(* Logix 5000 project; controller Week_4_PLC_1_Compare_Instructions Emulate 5570 rev 30.11; software revision 30.01 *)

TASK MainTask (continuous, watchdog 500 ms) : MainProgram

MODULES
   Local : Emulate 5570 (ICP 2, rev 30.11)
END_MODULES

PROGRAM MainProgram   (* main routine MainRoutine *)
VAR
   Counter : COUNTER := (PRE := 10);
   Output1 : BOOL;
   Output2 : BOOL;
   Output3 : BOOL;
   Output4 : BOOL;
   Output5 : BOOL;
   PB1 : BOOL;
END_VAR

ROUTINE MainRoutine   (* ladder *)
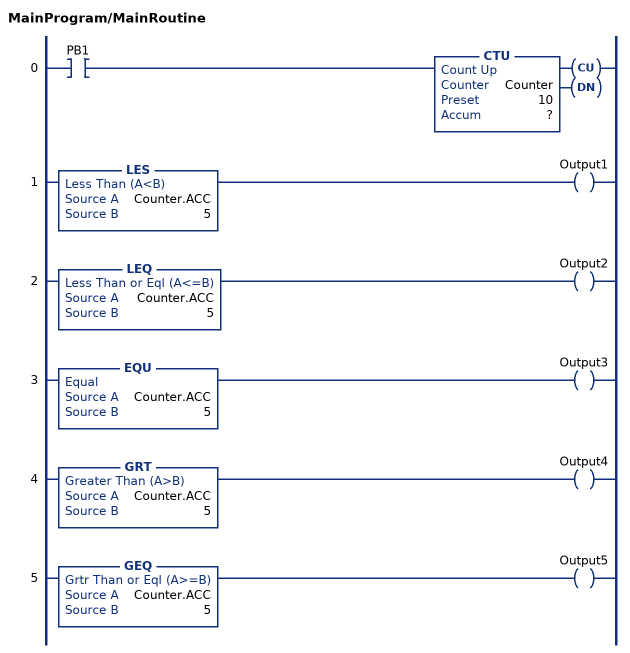
   0: XIC(PB1)CTU(Counter,?,?);
   1: LES(Counter.ACC,5)OTE(Output1);
   2: LEQ(Counter.ACC,5)OTE(Output2);
   3: EQU(Counter.ACC,5)OTE(Output3);
   4: GRT(Counter.ACC,5)OTE(Output4);
   5: GEQ(Counter.ACC,5)OTE(Output5);
END_ROUTINE
END_PROGRAM
